{attribute 'GeneratedUsingTerminal: EL7221-0001-0021'}
{attribute addProperty BoxType "EL7221-0001-0021"}
{attribute addProperty Description "EL7221-0001 1Ch. DS402 Servo motor output stage (50V, 8A RMS)"}
{attribute addProperty Physics "KK"}
{attribute addProperty Id "DS402_StatuswordAT %I*DS402_Statusword_9B36FDFC2DS402_Position_actual_valueAT %I*DS402_Position_actual_value_07DC4C744DS402_ControlwordAT %Q*DS402_Controlword_F3F147212DS402_Target_velocityAT %Q*DS402_Target_velocity_08A9583B4WcStateAT %I*WcState_9091E0EB2InfoDataAT %I*InfoData_96C94FAE19"}
{attribute addProperty CRC "2079462167"}
{attribute addProperty Size "33"}
TYPE EL7221_7BF21317 EXTENDS EtcSlaveTerminalBase_947E5A46 :
STRUCT
	{attribute addProperty Name "DS402_Statusword"}
	DS402_Statusword : DS402_Statusword_9B36FDFC;
	{attribute addProperty Name "DS402_Position_actual_value"}
	DS402_Position_actual_value : DS402_Position_actual_value_07DC4C74;
	{attribute addProperty Name "DS402_Controlword"}
	DS402_Controlword : DS402_Controlword_F3F14721;
	{attribute addProperty Name "DS402_Target_velocity"}
	DS402_Target_velocity : DS402_Target_velocity_08A9583B;
	{attribute addProperty Name "WcState"}
	WcState : WcState_9091E0EB;
	{attribute addProperty Name "InfoData"}
	InfoData : InfoData_96C94FAE;
END_STRUCT
END_TYPE

(* stored: Version 1.2.0.0, ProductVersion 3.1.4024.11
   DUT EL7221_7BF21317: Id {9847aba0-8da2-4e10-bd2f-6f4569a4d60a} *)
